// TIA Portal V20 export
DATA_BLOCK "Adatok_G2"   // DB2
{ S7_Optimized_Access := 'TRUE' }
// stored: MemoryReserve 100
BEGIN
END_DATA_BLOCK
